FUNCTION_BLOCK AnyTypeTest EXTENDS TcUnit.FB_TestSuite
VAR_INPUT
END_VAR
VAR_OUTPUT
END_VAR
VAR
END_VAR

CheckIsAnyTypeBinded();
ReturnsValidAnyType();

METHOD CheckIsAnyTypeBinded 
VAR
	expected : BOOL;
	actual : BOOL;
	isOpen : BOOL;
	anyBound : __SYSTEM.AnyType; 
END_VAR
TcUnit.TEST('isAnyTypeBinded should correctly detect binding state of ANYTYPE');

// --- Case 1: Unbound ANYTYPE ---
anyBound.diSize :=0;
anyBound.pValue :=0;
  
AssertEquals_BOOL(
	Expected := FALSE,
	Actual   := isAnyTypeBinded(anyType := anyBound),
	Message  := 'Expected FALSE when ANYTYPE.pValue = 0 and diSize = 0 (unbound)');
	
// --- Case 2: Bound ANYTYPE ---
anyBound.pValue :=	ADR(isOpen);
anyBound.diSize := SIZEOF(isOpen);
  
AssertEquals_BOOL(
	Expected := TRUE,
	Actual   := isAnyTypeBinded(anyType := anyBound),
	Message  := 'Expected TRUE when ANYTYPE.pValue is valid and diSize > 0 (bound)');

TEST_FINISHED();
END_METHOD

METHOD ReturnsValidAnyType
VAR
	expected : BOOL;
	actual : BOOL;
	
	intValue : INT;
	returnOfAnyType : __SYSTEM.AnyType;
	ptrOk  : BOOL;
	sizeOk : BOOL;  
END_VAR
TcUnit.TEST('ToAnyType should return a valid __SYSTEM.AnyType when passed an INT value');

returnOfAnyType := ToAnyType(intValue);

ptrOk := returnOfAnyType.pValue<>0;
sizeOk := returnOfAnyType.diSize = SIZEOF(intValue);

expected := TRUE;
actual := ptrOk AND sizeOk;

AssertEquals(
	Expected := expected,
	Actual   := actual,
	Message  := 'ToAnyType() failed: pValue was 0 or diSize was incorrect for INT input.');
	
TEST_FINISHED();
END_METHOD

END_FUNCTION_BLOCK

(* stored: Version 1.1.0.1, ProductVersion 3.1.4024.12
   POU AnyTypeTest: Id {98942519-e7b3-00c7-39b8-4b53b9a409c5}, SpecialFunc None
   Method CheckIsAnyTypeBinded: Id {63f30f07-1320-0063-3593-046d0d959e15}
   Method ReturnsValidAnyType: Id {f0d6fb56-3d24-0d3d-291b-e7133c3a727c} *)
